FUNCTION_BLOCK xPPU_SSC
VAR_INPUT
	i_error: POINTER TO ErrorManager;
	i_process: POINTER TO ProcessManager;
	i_state: POINTER TO StateTracker;
END_VAR
VAR
	m_emptyParams: ParameterSet;
	m_subRes: EOperationResult;
END_VAR

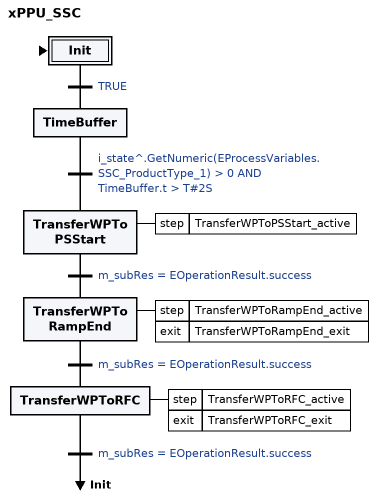
INITIAL_STEP Init:
END_STEP
TRANSITION FROM Init TO TimeBuffer
    := TRUE;
END_TRANSITION
STEP TimeBuffer:
END_STEP
TRANSITION FROM TimeBuffer TO TransferWPToPSStart
    := i_state^.GetNumeric(EProcessVariables.SSC_ProductType_1) > 0 AND TimeBuffer.t > T#2S;
END_TRANSITION
STEP TransferWPToPSStart:
    TransferWPToPSStart_active(N);  // step action
END_STEP
TRANSITION FROM TransferWPToPSStart TO TransferWPToRampEnd
    := m_subRes = EOperationResult.success;
END_TRANSITION
STEP TransferWPToRampEnd:
    TransferWPToRampEnd_active(N);  // step action
    TransferWPToRampEnd_exit(P0);  // exit action
END_STEP
TRANSITION FROM TransferWPToRampEnd TO TransferWPToRFC
    := m_subRes = EOperationResult.success;
END_TRANSITION
STEP TransferWPToRFC:
    TransferWPToRFC_active(N);  // step action
    TransferWPToRFC_exit(P0);  // exit action
END_STEP
TRANSITION FROM TransferWPToRFC TO Init
    := m_subRes = EOperationResult.success;
END_TRANSITION

ACTION TransferWPToPSStart_active:
m_subRes := i_process^.Execute(
	EBehaviorType.control_primitive,
	EPrimitives.SSC_TransferWorkpieceTo_PSStart,
	m_emptyParams);
END_ACTION

ACTION TransferWPToRampEnd_active:
m_subRes := i_process^.Execute(
	EBehaviorType.control_primitive,
	EPrimitives.SSC_TransferWorkpieceTo_RampEnd,
	m_emptyParams);
END_ACTION

ACTION TransferWPToRampEnd_exit:
i_state^.ShiftProduct(EProducts.SSC_product1,0);
END_ACTION

ACTION TransferWPToRFC_active:
m_subRes := i_process^.Execute(
	EBehaviorType.control_primitive,
	EPrimitives.SSC_TransferWorkpieceTo_RFC,
	m_emptyParams);
END_ACTION

ACTION TransferWPToRFC_exit:
i_state^.ShiftProduct(EProducts.SSC_product1, EProducts.RFC_product1);
i_state^.ShiftProduct(EProducts.SSC_product2, EProducts.RFC_product2);
END_ACTION

END_FUNCTION_BLOCK

(* stored: Version 1.1.0.1
   POU xPPU_SSC: Id {4ca0c2fa-6b16-48bd-a71d-fd301fc31cc7}, SpecialFunc None
   Action TransferWPToPSStart_active: Id {b3acd69f-0255-4601-91c6-2ba0e00b22e5}
   Action TransferWPToRampEnd_active: Id {51144d9b-8e79-4a05-9453-918c572208e0}
   Action TransferWPToRampEnd_exit: Id {7d7f48dd-f07a-4992-85cb-262e470b1b85}
   Action TransferWPToRFC_active: Id {53025564-8a58-4c33-bc47-c1de6154343e}
   Action TransferWPToRFC_exit: Id {f9cdcadb-df53-4921-84b7-a57c10cc748e} *)
